PROGRAM P_SequenceReader
VAR
END_VAR

//best effort servo follower.
//Elapsed time
//each time signature gets a value in mm for it's position relative to the 0 point of the system.
//buffer 3 seconds worth of data?

END_PROGRAM

(* stored: Version 1.1.0.1, ProductVersion 3.1.4024.3
   POU P_SequenceReader: Id {b7f6e06f-02ce-4bed-9da9-aa8070aed894}, SpecialFunc None *)
